Staubli VAL3: delete.pgx

public program delete(string x_sName, num& x_nResult[])
  local string l_sItem
  local num l_nSize
  local string l_sMessage
begin
  //
  // delete the select trajectory
  //
  if isDefined(pt:tTraj[x_sName]) and x_sName!="home"
    // delete
    delete(pt:tTraj[x_sName])
    // save it
    bToSave=true
    x_nResult=0
  elseIf x_sName=="home"
    call language:message(l_sMessage,133)
    popUpMsg(l_sMessage)
  else
    x_nResult=-1
  endIf
end
